(* CoDeSys 2.3.9.37 project: Cap11_4.pro *)
(* Libraries: Standard.lib 4.10.05 12:14:46, IecSfc.lib 13.4.06 16:51:28 *)

(* POU PLC_PRG, SFC *)
PROGRAM PLC_PRG
VAR
      (* Entradas *)
	A: BOOL;
	B: BOOL;
	Control: BOOL;
	(*Salidas*)
	Salida: BOOL;
	(*Otras*)
	MiTempo: TON;
END_VAR
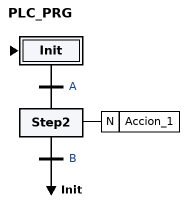
INITIAL_STEP Init:
END_STEP
TRANSITION FROM Init TO Step2 := A;
END_TRANSITION
STEP Step2:
	Accion_1(N);
END_STEP
TRANSITION FROM Step2 TO Init := B;
END_TRANSITION
END_PROGRAM
ACTION Accion_1:
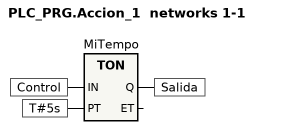
_FBD_ (* Function Block Diagram *)
NETWORK 1
	MiTempo:TON(IN: Control, PT: T#5s) => Salida
_END_FBD_
(* the same logic as Structured Text *)
(* Network 1 *)
MiTempo(IN := Control, PT := T#5s);
Salida := MiTempo.Q;
END_ACTION

(* Visualisation Visu
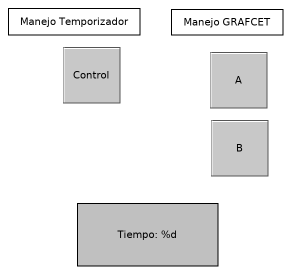
button at (80,54)-(137,110): text "Control"; toggles PLC_PRG.Control
button at (227,59)-(284,115): text "A"; taps PLC_PRG.A
button at (228,127)-(285,183): text "B"; taps PLC_PRG.B
rectangle at (25,15)-(157,42): text "Manejo Temporizador"
rectangle at (188,16)-(300,42): text "Manejo GRAFCET"
rounded rectangle at (94,210)-(235,273): text "Tiempo: %d"; shows PLC_PRG.MiTempo.ET; alarm colour if PLC_PRG.Salida
*)
